# EPICS substitutions: db/ecmcEL4122.substitutions
file ecmcEL4XXX-chX.template
{
	pattern {CH_ID, LINR,    ESLO,          EOFF,   EGU,     PREC, LOW, LOLO, HIGH, HIHI, HYST, LLSV,       LSV,        HSV,        HHSV      }
		{1,     "SLOPE", 4.882961516E-4,  4,      "mA",    0,    0,   0,    0,    0,    0,    "NO_ALARM", "NO_ALARM", "NO_ALARM", "NO_ALARM"}
		{2,     "SLOPE", 4.882961516E-4,  4,      "mA",    0,    0,   0,    0,    0,    0,    "NO_ALARM", "NO_ALARM", "NO_ALARM", "NO_ALARM"}
}
